Staubli VAL3: OnF2.pgx

program OnF2()
begin
  switch nPage
    //
    case 0
      call Offset(trOffset)
      libSave()
    break
    //
    case 1
      disablePower()
      resetMotion()
      call killAllTask()
      nPage=0
      bExit=true
    break
  endSwitch
  bUserRefresh=true
end
